(* PLC project TC3_TE1400_GeneratedModule_AdaptiveModel_FB, Beckhoff Automation GmbH & Co. KG TwinCAT 3 Function - TE1400 1.2.1240 *)
(* stored: companyURL www.beckhoff.com, creationDateTime 2022-01-04T00:47:12 *)

TYPE E_TcMatSimDataAreaType : (NotSpecified := 0, Standard, InputSrc, InputDst, OutputSrc, OutputDst, InternalDa, MArea, RetainDa);
END_TYPE

TYPE ST_TcMatSimObjectDataAreaInfo : STRUCT
  pPlcVar : PVOID;
  pModuleProcImg : PVOID;
  nSize : UDINT;
  nDataAreaId : UDINT;
  eDataAreaType : E_TcMatSimDataAreaType;
END_STRUCT;
END_TYPE

{attribute 'pack_mode' := '4'}
TYPE ST_AdaptiveModelInitData : STRUCT
  Header : TComInitDataHdr;
  CallByHdr : TComInitDataElmHdr;
  CallBy : TctModuleCallByType;
  ExecutionSequenceHdr : TComInitDataElmHdr;
  ExecutionSequence : TctModuleExecutionSequenceType;
  StepSizeHdr : TComInitDataElmHdr;
  StepSize : TctStepSizeType;
  ExecuteModelCodeHdr : TComInitDataElmHdr;
  ExecuteModelCode : BOOL;
  ModelParametersHdr : TComInitDataElmHdr;
  ModelParameters : P_AdaptiveModel_T;
  ContextInfoArr_0_TaskOidHdr : TComInitDataElmHdr;
  ContextInfoArr_0_TaskOid : OTCID;
  ContextInfoArr_0_TaskPriorityHdr : TComInitDataElmHdr;
  ContextInfoArr_0_TaskPriority : UDINT;
  ContextInfoArr_0_TaskCycleTimeNsHdr : TComInitDataElmHdr;
  ContextInfoArr_0_TaskCycleTimeNs : UDINT;
  ContextInfoArr_0_TaskPortHdr : TComInitDataElmHdr;
  ContextInfoArr_0_TaskPort : UINT;
  ContextInfoArr_0_TaskSortOrderHdr : TComInitDataElmHdr;
  ContextInfoArr_0_TaskSortOrder : UDINT;
END_STRUCT;
END_TYPE

TYPE ST_AdaptiveModel_Input : STRUCT
  In1 : LREAL;
END_STRUCT;
END_TYPE

TYPE ST_AdaptiveModel_Output : STRUCT
  Out1 : LREAL;
END_STRUCT;
END_TYPE

FUNCTION_BLOCK FB_TcMatSimObject
  VAR_INPUT
    bWriteFbInputValues : BOOL := TRUE;  (* set this flag to write FB input values to the TcComObject's input DataAreas. This will overwrite the mapped input values before module execution. Set to FALSE to read the mapped input values from the TcComObject to the FB. *)
  END_VAR
  VAR
    pDataAreas : POINTER TO ST_TcMatSimObjectDataAreaInfo;  (* process image src and dst pointers and sizes *)
    nDataAreas : UDINT;
    ipObjSrv : ITComObjectServer;  (* global interface pointers *)
    ipTcComObj : ITComObject;  (* object interface pointers *)
    ipTcCyclic : ITcCyclic;
    ipTcPostCyclic : ITcPostCyclic;
    ipTcAdi : ITcADI;
    ipTask : ITcTask;  (* task interface pointers *)
    pInitData : POINTER TO TComInitDataHdr;  (* initial parameters *)
    hResult : HRESULT;  (* hResult of interface calls (0 if no error) *)
    moduleClsId : CLSID;  (* module class ID *)
    assignedClsId : CLSID;  (* expected/desired module class ID *)
    bClassIdVerified : BOOL;
    bDynInstance : BOOL;  (* flag indicating whether the module instance was created dynamically *)
    eInitialObjState : TCOM_STATE := TCOM_STATE.TCOM_STATE_INIT;  (* the object state at the time FB_init was called, FB_exit will try to switch to this state (only if this means to shift down) *)
  END_VAR

            
          

{attribute 'object_name' := 'ReleaseTcComInterface'}
METHOD ReleaseTcComInterface : HRESULT
  VAR
    nStateChangeCnt : DINT := 0;
  END_VAR
                  
IF (ipTcComObj<>0) THEN
  WHILE (State>eInitialObjState AND nStateChangeCnt<1000) DO
    State := eInitialObjState;
    nStateChangeCnt := nStateChangeCnt+1;
  END_WHILE
  ReleaseObjInterfaces();
  IF (bDynInstance) THEN
    ReleaseTcComInterface := TC3_MODULE.FW_ObjMgr_DeleteInstance(ADR(ipTcComObj));
  ELSE
    ipTcComObj.TcRelease();
  END_IF
  ipTcComObj := 0;
END_IF
                  
                
END_METHOD

{attribute 'object_name' := 'ReleaseObjInterfaces'}
METHOD ReleaseObjInterfaces : HRESULT
                  
// release interface pointers
IF (ipTcCyclic<>0) THEN
  ipTcCyclic.TcRelease();
  ipTcCyclic := 0;
END_IF
IF (ipTcPostCyclic<>0) THEN
  ipTcPostCyclic.TcRelease();
  ipTcPostCyclic := 0;
END_IF
IF (ipTcAdi<>0) THEN
  ipTcAdi.TcRelease();
  ipTcAdi := 0;
END_IF
                  
                
END_METHOD

{attribute 'object_name' := 'Internal_SetObjState'}
METHOD Internal_SetObjState
  VAR_INPUT
    hr : REFERENCE TO HRESULT;
    nextState : TCOM_STATE;
  END_VAR
                  
// verify class id
IF (SUCCEEDED(hr)) THEN
  hr := VerifyClassId();
END_IF

// switch object state
IF (SUCCEEDED(hr) AND nextState>=TCOM_STATE_INIT) THEN
  IF (ipTcComObj=0) THEN
    hr := Tc2_System.E_HRESULTAdsErr.NOINTERFACE;
  END_IF
  IF (ipObjSrv=0) THEN
    hr := Tc2_System.E_HRESULTAdsErr.NOINTERFACE;
  END_IF
  IF (SUCCEEDED(hr)) THEN
    hr := ipTcComObj.TcSetObjState(nextState,ipObjSrv,pInitData);
  END_IF
END_IF
                  
                
END_METHOD

{attribute 'object_name' := 'FB_init'}
METHOD FB_init : BOOL
  VAR_INPUT
    bInitRetains : BOOL;  (* init retain variables *)
    bInCopyCode : BOOL;  (* Online Change *)
    oid : OTCID;
  END_VAR
                  
FB_init := SUCCEEDED(Init(oid));
                  
                
END_METHOD

{attribute 'object_name' := 'GetObjPara'}
METHOD GetObjPara : HRESULT
  VAR_INPUT
    pid : PTCID;
    nData : UDINT;
    pData : PVOID;
  END_VAR
                  
IF (ipTcComObj=0) THEN
  GetObjPara := Tc2_System.E_HRESULTAdsErr.NOINTERFACE;
END_IF

IF (SUCCEEDED(GetObjPara)) THEN
  GetObjPara := ipTcComObj.TcGetObjPara(pid:=pid,nData,pData,0);
END_IF
                  
                
END_METHOD

{attribute 'object_name' := 'QueryObjInterface'}
METHOD QueryObjInterface
  VAR_INPUT
    hr : REFERENCE TO HRESULT;
    iid : REFERENCE TO IID;
    pipItf : POINTER TO ITcUnknown;
  END_VAR
  VAR CONSTANT
    pNull : PVOID := 0;
  END_VAR
                  
IF (SUCCEEDED(hr)) THEN
  IF (ipTcComObj=0) THEN
    hr := Tc2_System.E_HRESULTAdsErr.NOINTERFACE;
  ELSIF (pipItf^=ULINT_TO_DWORD(pNull)) THEN
    hr := ipTcComObj.TcQueryInterface(iid:= iid, pipItf:=pipItf);
  END_IF
END_IF
                  
                
END_METHOD

{attribute 'object_name' := 'SaveOnlineParametersForInit'}
METHOD SaveOnlineParametersForInit : HRESULT
  VAR
    idx : UINT;
    pInitElemHdr : POINTER TO TComInitDataElmHdr;
    pData : PVOID;
    nData : UDINT;
  END_VAR
  VAR CONSTANT
    nInitDataAlignment : UDINT := 4;
  END_VAR
                  IF (pInitData<>0) THEN
  pInitElemHdr := pInitData + SIZEOF(pInitData^);
  FOR idx:=1 TO pInitData^.uiElmCnt DO
    pData := pInitElemHdr + ULINT_TO_DWORD(SIZEOF(pInitElemHdr^));
    nData := pInitElemHdr^.cbData;
    SaveOnlineParametersForInit := GetObjPara(pInitElemHdr^.indexOffset,nData,pData);
    IF (FAILED(SaveOnlineParametersForInit)) THEN
      RETURN;
    END_IF
    pInitElemHdr := pData + (nInitDataAlignment*((nData + nInitDataAlignment - 1)/nInitDataAlignment));
  END_FOR
ELSE
	SaveOnlineParametersForInit := Tc2_System.E_HRESULTAdsErr.NOTINIT;
END_IF
                  
                
END_METHOD

{attribute 'object_name' := 'ResetHresult'}
METHOD ResetHresult
                  hResult := S_OK;
                
END_METHOD

{attribute 'object_name' := 'Execute'}
METHOD Execute : HRESULT
  VAR
    nDaIdx : UDINT;
    pCurDataArea : POINTER TO ST_TcMatSimObjectDataAreaInfo;
  END_VAR
                  
IF (SUCCEEDED(hResult)) THEN
  hResult := VerifyClassId();
END_IF

IF (SUCCEEDED(hResult) AND State<>TCOM_STATE_OP) THEN
  hResult := Tc2_System.E_HRESULTAdsErr.NOTREADY;
END_IF

// get image pointers
IF (SUCCEEDED(hResult)) THEN
  GetImagePtrs(hResult);
END_IF

// copy inputs
IF (pDataAreas<>0 AND nDataAreas>0 AND bWriteFbInputValues) THEN
  FOR nDaIdx:=0 TO nDataAreas-1 DO
    IF (FAILED(hResult))THEN
      CONTINUE;
    END_IF
    pCurDataArea := pDataAreas + nDaIdx*SIZEOF(ST_TcMatSimObjectDataAreaInfo);
    IF ((pCurDataArea^.eDataAreaType <> E_TcMatSimDataAreaType.InputDst))THEN
      CONTINUE;
    END_IF
    IF (pCurDataArea^.pModuleProcImg<>0 AND pCurDataArea^.pPlcVar<>0) THEN
      MEMCPY(pCurDataArea^.pModuleProcImg,pCurDataArea^.pPlcVar,pCurDataArea^.nSize);
    ELSE
      hResult := Tc2_System.E_HRESULTAdsErr.NOINTERFACE;
    END_IF
  END_FOR
END_IF

// call cycle update
IF (SUCCEEDED(hResult)) THEN
  IF (ipTcCyclic<>0) THEN
    hResult := ipTcCyclic.CycleUpdate(ipTask:= ipTask, ipCaller:= 0, context:= 0);
  ELSE
    hResult := Tc2_System.E_HRESULTAdsErr.NOINTERFACE;
  END_IF
END_IF

// copy outputs
IF (pDataAreas<>0 AND nDataAreas>0) THEN
  FOR nDaIdx:=0 TO nDataAreas-1 DO
    IF (FAILED(hResult))THEN
      CONTINUE;
    END_IF
    pCurDataArea := pDataAreas + nDaIdx*SIZEOF(ST_TcMatSimObjectDataAreaInfo);
    IF ((pCurDataArea^.eDataAreaType = E_TcMatSimDataAreaType.OutputSrc) OR NOT bWriteFbInputValues) THEN
      IF (pCurDataArea^.pModuleProcImg<>0 AND pCurDataArea^.pPlcVar<>0) THEN
        MEMCPY(pCurDataArea^.pPlcVar,pCurDataArea^.pModuleProcImg,pCurDataArea^.nSize);
      ELSE
        hResult := Tc2_System.E_HRESULTAdsErr.NOINTERFACE;
      END_IF
    END_IF
  END_FOR
END_IF


// call post cyclic update
IF (SUCCEEDED(hResult)) THEN
  IF (ipTcPostCyclic<>0) THEN
    hResult := ipTcPostCyclic.PostCyclicUpdate(ipTask:= 0, ipCaller:= 0, context:= 0);
  ELSE
    hResult := Tc2_System.E_HRESULTAdsErr.NOINTERFACE;
  END_IF
END_IF

ReleaseImagePtrs();

Execute := hResult;
                  
                
END_METHOD

{attribute 'object_name' := 'GetImagePtrs'}
METHOD GetImagePtrs
  VAR_INPUT
    hr : REFERENCE TO HRESULT;
  END_VAR
  VAR
    nDaIdx : UDINT;
    pCurDataArea : POINTER TO ST_TcMatSimObjectDataAreaInfo;
  END_VAR
                  
IF (ipTcAdi=0) THEN
  hr := Tc2_System.E_HRESULTAdsErr.NOINTERFACE;
END_IF
IF(State<>TCOM_STATE_OP)THEN
  hr := Tc2_System.E_HRESULTAdsErr.INVALIDSTATE;
END_IF


// get pointers to process images
IF (pDataAreas<>0 AND nDataAreas>0) THEN
  FOR nDaIdx:=0 TO nDataAreas-1 DO
    pCurDataArea := pDataAreas + nDaIdx*SIZEOF(ST_TcMatSimObjectDataAreaInfo);
    IF (FAILED(hr))THEN
      CONTINUE;
    END_IF
    IF ((pCurDataArea^.eDataAreaType <> E_TcMatSimDataAreaType.InputDst) AND (pCurDataArea^.eDataAreaType <> E_TcMatSimDataAreaType.OutputSrc))THEN
      CONTINUE;
    END_IF
    IF (pCurDataArea^.pModuleProcImg=0 AND pCurDataArea^.nSize>0) THEN
      hr := ipTcAdi.GetImagePtr(size:= pCurDataArea^.nSize , offs:=0 , adi_x:=pCurDataArea^.nDataAreaId , ppData:=ADR(pCurDataArea^.pModuleProcImg));
    END_IF
  END_FOR
END_IF

IF (FAILED(hr)) THEN
  ReleaseImagePtrs();
END_IF
                  
                
END_METHOD

{attribute 'object_name' := 'VerifyClassId'}
METHOD VerifyClassId : HRESULT
  VAR
    emptyClsId : CLSID;
  END_VAR
                  memset(ADR(emptyClsId),0,SIZEOF(emptyClsId));
IF (bClassIdVerified) THEN
  // class ID was already verified
  VerifyClassId := Tc2_System.E_HRESULTAdsErr.HRESULT_ADS_NOERROR;
ELSIF (memcmp(ADR(assignedClsId),ADR(emptyClsId),SIZEOF(assignedClsId))=0) THEN
  // skip class ID verification if no assignedClsId specified
  VerifyClassId := Tc2_System.E_HRESULTAdsErr.HRESULT_ADS_NOERROR;
ELSE
  // verify class ID
  VerifyClassId := ReadModuleClassId();

  IF (SUCCEEDED(VerifyClassId)) THEN
    IF (memcmp(ADR(assignedClsId),ADR(moduleClsId),SIZEOF(assignedClsId))<>0) THEN
     VerifyClassId := Tc2_System.E_HRESULTAdsErr.INVALIDCLSID;
    END_IF
  END_IF
  bClassIdVerified := SUCCEEDED(VerifyClassId);
END_IF
                  
                
END_METHOD

{attribute 'object_name' := 'SetObjPara'}
METHOD SetObjPara : HRESULT
  VAR_INPUT
    pid : PTCID;
    nData : UDINT;
    pData : PVOID;
  END_VAR
                  
IF (ipTcComObj=0) THEN
  SetObjPara := Tc2_System.E_HRESULTAdsErr.NOINTERFACE;
END_IF

IF (SUCCEEDED(SetObjPara)) THEN
  SetObjPara := ipTcComObj.TcSetObjPara(pid:=pid,nData,pData,0);
END_IF
                  
                
END_METHOD

{attribute 'object_name' := 'QueryTcComInterface'}
METHOD QueryTcComInterface
  VAR_INPUT
    hr : REFERENCE TO HRESULT;
    oid : OTCID;
  END_VAR
                  
IF (ipObjSrv=0) THEN
  hr := Tc2_System.E_HRESULTAdsErr.NOINTERFACE;
END_IF

IF (SUCCEEDED(hr) AND ipTcComObj=0) THEN
  bDynInstance := FALSE;
  IF(oid>0) THEN
    // query interface of existing object
    hr := ipObjSrv.TcQueryObjectInterface(oid,IID_ITComObject,ADR(ipTcComObj));
  ELSE
    // create new instance and get the object interface
    hr := ipObjSrv.TcCreateInstance(assignedClsId,IID_ITComObject,ADR(ipTcComObj));
    IF (SUCCEEDED(hr)) THEN
      bDynInstance := TRUE;
      hr := ipTcComObj.TcSetObjectId(OTCID_CreateNewId);
    END_IF
  END_IF
  IF (SUCCEEDED(hr)) THEN
    eInitialObjState := State;
  END_IF
END_IF
                  
                
END_METHOD

{attribute 'object_name' := 'ReleaseImagePtrs'}
METHOD ReleaseImagePtrs : HRESULT
  VAR
    nDaIdx : UDINT;
    pCurDataArea : POINTER TO ST_TcMatSimObjectDataAreaInfo;
  END_VAR
                  
IF (ipTcAdi=0) THEN
  ReleaseImagePtrs := Tc2_System.E_HRESULTAdsErr.NOINTERFACE;
END_IF

IF (SUCCEEDED(ReleaseImagePtrs) AND pDataAreas<>0 AND nDataAreas>0) THEN
  // release pointers to the simulink module process images
  FOR nDaIdx:=0 TO nDataAreas-1 DO
    pCurDataArea := pDataAreas + nDaIdx*SIZEOF(ST_TcMatSimObjectDataAreaInfo);

    IF (pCurDataArea^.pModuleProcImg<>0) THEN
      ipTcAdi.ReleaseImagePtr(pData:=pCurDataArea^.pModuleProcImg);
      pCurDataArea^.pModuleProcImg := 0;
    END_IF
  END_FOR
END_IF
                  
                
END_METHOD

{attribute 'object_name' := 'FB_exit'}
METHOD FB_exit : BOOL
  VAR_INPUT
    bInCopyCode : BOOL;  (* Online Change *)
  END_VAR
                  
IF (NOT bInCopyCode) THEN
  IF (ipObjSrv<>0) THEN
    ipObjSrv.TcRelease();
    ipObjSrv := 0;
  END_IF

  ReleaseTcComInterface();
END_IF
                  
                
END_METHOD

{attribute 'object_name' := 'InitObjName'}
METHOD InitObjName
  VAR_INPUT
    hr : REFERENCE TO HRESULT;
  END_VAR
  VAR
    objectName : STRING(255) := 'TcMatSimObject_PlcRtFbInstance';
    oid : OTCID;
  END_VAR
                  
IF (SUCCEEDED(hr)) THEN
  hr := ipTcComObj.TcGetObjectId(oid);
END_IF

IF (SUCCEEDED(hr) and bDynInstance) THEN
  objectName := TC2_STANDARD.CONCAT(objectName,'_');
  objectName := TC2_STANDARD.CONCAT(objectName,UDINT_TO_STRING(oid));
  hr := ipTcComObj.TcSetObjectName(ADR(objectName));
END_IF
                  
                
END_METHOD

{attribute 'object_name' := 'SetObjState'}
METHOD SetObjState : HRESULT
  VAR_INPUT
    finalState : TCOM_STATE;
  END_VAR
  VAR
    bShiftUp : BOOL;
    bShiftDown : BOOL;
    currentState : TCOM_STATE;
  END_VAR
                  
currentState := State;

bShiftUp := finalState>currentState;
bShiftDown := finalState<currentState;

// do not switch up on error
IF (FAILED(hresult)) THEN
  bShiftUp := FALSE;
END_IF
// reset existing error on switching down
IF (bShiftDown) THEN
  ResetHresult();
END_IF

// prepared state switch
CASE currentState OF
  TCOM_STATE_INIT:
    IF(bShiftUp) THEN
      QueryTcComInterface(hResult,0);
      Internal_SetObjState(hResult,TCOM_STATE.TCOM_STATE_PREOP);
      InitObjName(hResult);
    END_IF

  TCOM_STATE_PREOP:
    IF(bShiftUp) THEN
      Internal_SetObjState(hResult,TCOM_STATE.TCOM_STATE_SAFEOP);
      QueryObjInterfaces(hResult);
    ELSIF (bShiftDown) THEN
      Internal_SetObjState(hResult,TCOM_STATE.TCOM_STATE_INIT);
    END_IF

  TCOM_STATE_SAFEOP:
    IF(bShiftUp) THEN
      Internal_SetObjState(hResult,TCOM_STATE.TCOM_STATE_OP);
      QueryObjInterfaces(hResult);
    ELSIF (bShiftDown) THEN
      Internal_SetObjState(hResult,TCOM_STATE.TCOM_STATE_PREOP);
      ReleaseObjInterfaces();
    END_IF


  TCOM_STATE_OP:
    IF (bShiftDown) THEN
      Internal_SetObjState(hResult,TCOM_STATE.TCOM_STATE_SAFEOP);
    END_IF
END_CASE

SetObjState := hResult;
                  
                
END_METHOD

{attribute 'object_name' := 'QueryObjInterfaces'}
METHOD QueryObjInterfaces
  VAR_INPUT
    hr : REFERENCE TO HRESULT;
  END_VAR
                  
IF(State<TCOM_STATE_PREOP)THEN
  hr := Tc2_System.E_HRESULTAdsErr.INVALIDSTATE;
END_IF

//cyclic interface
QueryObjInterface(hr,IID_ITCCYCLIC,ADR(ipTcCyclic));
//post cyclic interface
QueryObjInterface(hr,IID_ITCPOSTCYCLIC,ADR(ipTcPostCyclic));
//adi interface
QueryObjInterface(hr,IID_ITcADI,ADR(ipTcAdi));
                  
                
END_METHOD

{attribute 'object_name' := 'Init'}
METHOD Init : HRESULT
  VAR_INPUT
    oid : OTCID;
  END_VAR
                  
// preinitialize variables
memset(ADR(moduleClsId),0,SIZEOF(moduleClsId));
bClassIdVerified := FALSE;
hResult := Tc2_System.E_HRESULTAdsErr.HRESULT_ADS_NOERROR;

// get object server
IF (ipObjSrv=0) THEN
  hResult := FW_ObjMgr_GetObjectServer(_AppInfo.ObjId,ADR(ipObjSrv));
END_IF

// try to get object interfaces
IF (SUCCEEDED(hresult)) THEN
  QueryTcComInterface(hResult,oid);
END_IF

// verify class id
IF (SUCCEEDED(hresult)) THEN
  hresult := VerifyClassId();
END_IF

// query interfaces, if the current state is higher than INIT
IF (SUCCEEDED(hresult) AND State>TCOM_STATE.TCOM_STATE_INIT) THEN
  QueryObjInterfaces(hResult);
END_IF

// return value
Init := hresult;
                  
                
END_METHOD

{attribute 'object_name' := 'ReadModuleClassId'}
METHOD ReadModuleClassId : HRESULT
  VAR
    emptyClsId : CLSID;
  END_VAR
                  memset(ADR(emptyClsId),0,SIZEOF(emptyClsId));
IF (memcmp(ADR(moduleClsId),ADR(emptyClsId),SIZEOF(moduleClsId))=0) THEN
  IF (ipTcComObj=0) THEN
    ReadModuleClassId := Tc2_System.E_HRESULTAdsErr.NOINTERFACE;
  END_IF

  //objectClsId := clsid;
  IF (SUCCEEDED(ReadModuleClassId)) THEN
    ReadModuleClassId := ipTcComObj.GetClassId(moduleClsId);
  END_IF
END_IF
                
END_METHOD

METHOD PUBLIC AssignClassId
VAR_INPUT
	clsId : CLSID;
END_VAR
                  assignedClsId := clsId;
bClassIdVerified := false;
                  
                
END_METHOD

PROPERTY Error : BOOL
GET
                    Error := FAILED(hResult);
                  
END_GET
END_PROPERTY

METHOD PUBLIC SetDataAreaInfo
VAR_INPUT
  pDataAreas: POINTER TO ST_TcMatSimObjectDataAreaInfo;
  nDataAreas: UDINT;
END_VAR
                  
THIS^.nDataAreas := nDataAreas;
THIS^.pDataAreas := pDataAreas;
                  
                
END_METHOD

METHOD PUBLIC SetInitDataInfo
VAR_INPUT
  pInitData : POINTER TO TComInitDataHdr;
END_VAR
                  this^.pInitData := pInitData;
                
END_METHOD

PROPERTY ClassId : CLSID
GET
                    hResult := ReadModuleClassId();
ClassId := moduleClsId;
                    
                  
END_GET
END_PROPERTY

PROPERTY State : TCOM_STATE
GET
  VAR
    hr : HRESULT := S_OK;
    eObjState : TCOM_STATE;
  END_VAR
                    
IF (ipTcComObj<>0) THEN
  hr := ipTcComObj.TcGetObjState(ADR(eObjState));
IF (FAILED(hr)) THEN
  eObjState := TCOM_STATE.TCOM_STATE_INIT;
END_IF
ELSE
  eObjState := TCOM_STATE.TCOM_STATE_INIT;
END_IF
State := eObjState;
                    
                  
END_GET
SET
                    SetObjState(State);
                  
END_SET
END_PROPERTY

PROPERTY ErrorCode : HRESULT
GET
                    ErrorCode := hResult;
                  
END_GET
END_PROPERTY
END_FUNCTION_BLOCK

{attribute 'TcDependOnClassFactory' := 'AdaptiveModel'}
FUNCTION_BLOCK FB_AdaptiveModel EXTENDS FB_TcMatSimObject
  VAR_INPUT
    stInput : ST_AdaptiveModel_Input;
  END_VAR
  VAR_OUTPUT
    stOutput : ST_AdaptiveModel_Output;
  END_VAR
  VAR
    stInitData : ST_AdaptiveModelInitData;
    arrDataAreas : ARRAY[1..2] OF ST_TcMatSimObjectDataAreaInfo;
    bParametersVerified : BOOL;
  END_VAR

            
          

{attribute 'object_name' := 'Internal_SetObjState'}
METHOD Internal_SetObjState
  VAR_INPUT
    hr : REFERENCE TO HRESULT;
    nextState : TCOM_STATE;
  END_VAR
                  
// update pointer to InitData structure
SetInitDataInfo(ADR(stInitData));
// call base method
SUPER^.Internal_SetObjState(hr,nextState);
                  
                
END_METHOD

{attribute 'object_name' := 'SaveOnlineParametersForInit'}
METHOD SaveOnlineParametersForInit : HRESULT
  VAR
    idx : UINT;
    pInitElemHdr : POINTER TO TComInitDataElmHdr;
    pData : PVOID;
    nData : UDINT;
  END_VAR
  VAR CONSTANT
    nInitDataAlignment : UDINT := 4;
  END_VAR
                  
// update pointer to InitData structure
SetInitDataInfo(ADR(stInitData));
// call base method
SaveOnlineParametersForInit := SUPER^.SaveOnlineParametersForInit();
                  
                
END_METHOD

METHOD FB_init : BOOL
  VAR_INPUT
    bInitRetains : BOOL;  (* if TRUE, the retain variables are initialized (warm start / cold start) *)
    bInCopyCode : BOOL;  (* if TRUE, the instance afterwards gets moved into the copy code (online change) *)
    oid : OTCID;
  END_VAR
  VAR
    clsId : CLSID;
  END_VAR
                  
// initialize flags
bParametersVerified := false;
                    
// set module class id for compatibility check
clsId.Data1 := 16#dc3905a3;
clsId.Data2 := 16#3c10;
clsId.Data3 := 16#463f;
clsId.Data4[0] := 16#97;
clsId.Data4[1] := 16#74;
clsId.Data4[2] := 16#0a;
clsId.Data4[3] := 16#63;
clsId.Data4[4] := 16#82;
clsId.Data4[5] := 16#3c;
clsId.Data4[6] := 16#f9;
clsId.Data4[7] := 16#4a;

AssignClassId(clsId);
                    
// initialize InitData structure with default values              
stInitData.CallByHdr.indexGroup := 0;
stInitData.CallByHdr.indexOffset := 16#00000000;
stInitData.CallByHdr.cbData := SIZEOF(stInitData.CallBy);
stInitData.CallBy := TctModuleCallByType.Module;
stInitData.ExecutionSequenceHdr.indexGroup := 0;
stInitData.ExecutionSequenceHdr.indexOffset := 16#00000001;
stInitData.ExecutionSequenceHdr.cbData := SIZEOF(stInitData.ExecutionSequence);
stInitData.ExecutionSequence := TctModuleExecutionSequenceType.StateUpdateAfterOutputMapping;
stInitData.StepSizeHdr.indexGroup := 0;
stInitData.StepSizeHdr.indexOffset := 16#00000002;
stInitData.StepSizeHdr.cbData := SIZEOF(stInitData.StepSize);
stInitData.StepSize := TctStepSizeType.RequireMatchingTaskCycleTime;
stInitData.ExecuteModelCodeHdr.indexGroup := 0;
stInitData.ExecuteModelCodeHdr.indexOffset := 16#00000007;
stInitData.ExecuteModelCodeHdr.cbData := SIZEOF(stInitData.ExecuteModelCode);
stInitData.ExecuteModelCode := 1;
stInitData.ModelParametersHdr.indexGroup := 0;
stInitData.ModelParametersHdr.indexOffset := 16#83000000;
stInitData.ModelParametersHdr.cbData := SIZEOF(stInitData.ModelParameters);
stInitData.ModelParameters.A_01 := 20;
stInitData.ModelParameters.a := 2;
stInitData.ModelParameters.b := 5;
stInitData.ModelParameters.DefuzzifyOutputs_SimulateUsing := 1;
stInitData.ModelParameters.EvaluateRuleAntecedents_Simulat := 1;
stInitData.ModelParameters.EvaluateRuleConsequents_Simulat := 1;
stInitData.ModelParameters.OutputSamplePoints_Value[0] := -6;
stInitData.ModelParameters.OutputSamplePoints_Value[1] := -6;
stInitData.ModelParameters.OutputSamplePoints_Value[2] := -6;
stInitData.ModelParameters.OutputSamplePoints_Value[3] := -5.8799999999999999;
stInitData.ModelParameters.OutputSamplePoints_Value[4] := -5.8799999999999999;
stInitData.ModelParameters.OutputSamplePoints_Value[5] := -5.8799999999999999;
stInitData.ModelParameters.OutputSamplePoints_Value[6] := -5.7599999999999998;
stInitData.ModelParameters.OutputSamplePoints_Value[7] := -5.7599999999999998;
stInitData.ModelParameters.OutputSamplePoints_Value[8] := -5.7599999999999998;
stInitData.ModelParameters.OutputSamplePoints_Value[9] := -5.6399999999999997;
stInitData.ModelParameters.OutputSamplePoints_Value[10] := -5.6399999999999997;
stInitData.ModelParameters.OutputSamplePoints_Value[11] := -5.6399999999999997;
stInitData.ModelParameters.OutputSamplePoints_Value[12] := -5.5199999999999996;
stInitData.ModelParameters.OutputSamplePoints_Value[13] := -5.5199999999999996;
stInitData.ModelParameters.OutputSamplePoints_Value[14] := -5.5199999999999996;
stInitData.ModelParameters.OutputSamplePoints_Value[15] := -5.4000000000000004;
stInitData.ModelParameters.OutputSamplePoints_Value[16] := -5.4000000000000004;
stInitData.ModelParameters.OutputSamplePoints_Value[17] := -5.4000000000000004;
stInitData.ModelParameters.OutputSamplePoints_Value[18] := -5.2800000000000002;
stInitData.ModelParameters.OutputSamplePoints_Value[19] := -5.2800000000000002;
stInitData.ModelParameters.OutputSamplePoints_Value[20] := -5.2800000000000002;
stInitData.ModelParameters.OutputSamplePoints_Value[21] := -5.1600000000000001;
stInitData.ModelParameters.OutputSamplePoints_Value[22] := -5.1600000000000001;
stInitData.ModelParameters.OutputSamplePoints_Value[23] := -5.1600000000000001;
stInitData.ModelParameters.OutputSamplePoints_Value[24] := -5.04;
stInitData.ModelParameters.OutputSamplePoints_Value[25] := -5.04;
stInitData.ModelParameters.OutputSamplePoints_Value[26] := -5.04;
stInitData.ModelParameters.OutputSamplePoints_Value[27] := -4.9199999999999999;
stInitData.ModelParameters.OutputSamplePoints_Value[28] := -4.9199999999999999;
stInitData.ModelParameters.OutputSamplePoints_Value[29] := -4.9199999999999999;
stInitData.ModelParameters.OutputSamplePoints_Value[30] := -4.7999999999999998;
stInitData.ModelParameters.OutputSamplePoints_Value[31] := -4.7999999999999998;
stInitData.ModelParameters.OutputSamplePoints_Value[32] := -4.7999999999999998;
stInitData.ModelParameters.OutputSamplePoints_Value[33] := -4.6799999999999997;
stInitData.ModelParameters.OutputSamplePoints_Value[34] := -4.6799999999999997;
stInitData.ModelParameters.OutputSamplePoints_Value[35] := -4.6799999999999997;
stInitData.ModelParameters.OutputSamplePoints_Value[36] := -4.5600000000000005;
stInitData.ModelParameters.OutputSamplePoints_Value[37] := -4.5600000000000005;
stInitData.ModelParameters.OutputSamplePoints_Value[38] := -4.5600000000000005;
stInitData.ModelParameters.OutputSamplePoints_Value[39] := -4.4399999999999995;
stInitData.ModelParameters.OutputSamplePoints_Value[40] := -4.4399999999999995;
stInitData.ModelParameters.OutputSamplePoints_Value[41] := -4.4399999999999995;
stInitData.ModelParameters.OutputSamplePoints_Value[42] := -4.3200000000000003;
stInitData.ModelParameters.OutputSamplePoints_Value[43] := -4.3200000000000003;
stInitData.ModelParameters.OutputSamplePoints_Value[44] := -4.3200000000000003;
stInitData.ModelParameters.OutputSamplePoints_Value[45] := -4.2000000000000002;
stInitData.ModelParameters.OutputSamplePoints_Value[46] := -4.2000000000000002;
stInitData.ModelParameters.OutputSamplePoints_Value[47] := -4.2000000000000002;
stInitData.ModelParameters.OutputSamplePoints_Value[48] := -4.0800000000000001;
stInitData.ModelParameters.OutputSamplePoints_Value[49] := -4.0800000000000001;
stInitData.ModelParameters.OutputSamplePoints_Value[50] := -4.0800000000000001;
stInitData.ModelParameters.OutputSamplePoints_Value[51] := -3.96;
stInitData.ModelParameters.OutputSamplePoints_Value[52] := -3.96;
stInitData.ModelParameters.OutputSamplePoints_Value[53] := -3.96;
stInitData.ModelParameters.OutputSamplePoints_Value[54] := -3.8399999999999999;
stInitData.ModelParameters.OutputSamplePoints_Value[55] := -3.8399999999999999;
stInitData.ModelParameters.OutputSamplePoints_Value[56] := -3.8399999999999999;
stInitData.ModelParameters.OutputSamplePoints_Value[57] := -3.7200000000000002;
stInitData.ModelParameters.OutputSamplePoints_Value[58] := -3.7200000000000002;
stInitData.ModelParameters.OutputSamplePoints_Value[59] := -3.7200000000000002;
stInitData.ModelParameters.OutputSamplePoints_Value[60] := -3.6000000000000001;
stInitData.ModelParameters.OutputSamplePoints_Value[61] := -3.6000000000000001;
stInitData.ModelParameters.OutputSamplePoints_Value[62] := -3.6000000000000001;
stInitData.ModelParameters.OutputSamplePoints_Value[63] := -3.48;
stInitData.ModelParameters.OutputSamplePoints_Value[64] := -3.48;
stInitData.ModelParameters.OutputSamplePoints_Value[65] := -3.48;
stInitData.ModelParameters.OutputSamplePoints_Value[66] := -3.3599999999999999;
stInitData.ModelParameters.OutputSamplePoints_Value[67] := -3.3599999999999999;
stInitData.ModelParameters.OutputSamplePoints_Value[68] := -3.3599999999999999;
stInitData.ModelParameters.OutputSamplePoints_Value[69] := -3.2400000000000002;
stInitData.ModelParameters.OutputSamplePoints_Value[70] := -3.2400000000000002;
stInitData.ModelParameters.OutputSamplePoints_Value[71] := -3.2400000000000002;
stInitData.ModelParameters.OutputSamplePoints_Value[72] := -3.1200000000000001;
stInitData.ModelParameters.OutputSamplePoints_Value[73] := -3.1200000000000001;
stInitData.ModelParameters.OutputSamplePoints_Value[74] := -3.1200000000000001;
stInitData.ModelParameters.OutputSamplePoints_Value[75] := -3;
stInitData.ModelParameters.OutputSamplePoints_Value[76] := -3;
stInitData.ModelParameters.OutputSamplePoints_Value[77] := -3;
stInitData.ModelParameters.OutputSamplePoints_Value[78] := -2.8799999999999999;
stInitData.ModelParameters.OutputSamplePoints_Value[79] := -2.8799999999999999;
stInitData.ModelParameters.OutputSamplePoints_Value[80] := -2.8799999999999999;
stInitData.ModelParameters.OutputSamplePoints_Value[81] := -2.7599999999999998;
stInitData.ModelParameters.OutputSamplePoints_Value[82] := -2.7599999999999998;
stInitData.ModelParameters.OutputSamplePoints_Value[83] := -2.7599999999999998;
stInitData.ModelParameters.OutputSamplePoints_Value[84] := -2.6400000000000001;
stInitData.ModelParameters.OutputSamplePoints_Value[85] := -2.6400000000000001;
stInitData.ModelParameters.OutputSamplePoints_Value[86] := -2.6400000000000001;
stInitData.ModelParameters.OutputSamplePoints_Value[87] := -2.52;
stInitData.ModelParameters.OutputSamplePoints_Value[88] := -2.52;
stInitData.ModelParameters.OutputSamplePoints_Value[89] := -2.52;
stInitData.ModelParameters.OutputSamplePoints_Value[90] := -2.3999999999999999;
stInitData.ModelParameters.OutputSamplePoints_Value[91] := -2.3999999999999999;
stInitData.ModelParameters.OutputSamplePoints_Value[92] := -2.3999999999999999;
stInitData.ModelParameters.OutputSamplePoints_Value[93] := -2.2799999999999998;
stInitData.ModelParameters.OutputSamplePoints_Value[94] := -2.2799999999999998;
stInitData.ModelParameters.OutputSamplePoints_Value[95] := -2.2799999999999998;
stInitData.ModelParameters.OutputSamplePoints_Value[96] := -2.1600000000000001;
stInitData.ModelParameters.OutputSamplePoints_Value[97] := -2.1600000000000001;
stInitData.ModelParameters.OutputSamplePoints_Value[98] := -2.1600000000000001;
stInitData.ModelParameters.OutputSamplePoints_Value[99] := -2.04;
stInitData.ModelParameters.OutputSamplePoints_Value[100] := -2.04;
stInitData.ModelParameters.OutputSamplePoints_Value[101] := -2.04;
stInitData.ModelParameters.OutputSamplePoints_Value[102] := -1.9199999999999999;
stInitData.ModelParameters.OutputSamplePoints_Value[103] := -1.9199999999999999;
stInitData.ModelParameters.OutputSamplePoints_Value[104] := -1.9199999999999999;
stInitData.ModelParameters.OutputSamplePoints_Value[105] := -1.7999999999999998;
stInitData.ModelParameters.OutputSamplePoints_Value[106] := -1.7999999999999998;
stInitData.ModelParameters.OutputSamplePoints_Value[107] := -1.7999999999999998;
stInitData.ModelParameters.OutputSamplePoints_Value[108] := -1.6799999999999997;
stInitData.ModelParameters.OutputSamplePoints_Value[109] := -1.6799999999999997;
stInitData.ModelParameters.OutputSamplePoints_Value[110] := -1.6799999999999997;
stInitData.ModelParameters.OutputSamplePoints_Value[111] := -1.5599999999999996;
stInitData.ModelParameters.OutputSamplePoints_Value[112] := -1.5599999999999996;
stInitData.ModelParameters.OutputSamplePoints_Value[113] := -1.5599999999999996;
stInitData.ModelParameters.OutputSamplePoints_Value[114] := -1.4400000000000004;
stInitData.ModelParameters.OutputSamplePoints_Value[115] := -1.4400000000000004;
stInitData.ModelParameters.OutputSamplePoints_Value[116] := -1.4400000000000004;
stInitData.ModelParameters.OutputSamplePoints_Value[117] := -1.3200000000000003;
stInitData.ModelParameters.OutputSamplePoints_Value[118] := -1.3200000000000003;
stInitData.ModelParameters.OutputSamplePoints_Value[119] := -1.3200000000000003;
stInitData.ModelParameters.OutputSamplePoints_Value[120] := -1.2000000000000002;
stInitData.ModelParameters.OutputSamplePoints_Value[121] := -1.2000000000000002;
stInitData.ModelParameters.OutputSamplePoints_Value[122] := -1.2000000000000002;
stInitData.ModelParameters.OutputSamplePoints_Value[123] := -1.0800000000000001;
stInitData.ModelParameters.OutputSamplePoints_Value[124] := -1.0800000000000001;
stInitData.ModelParameters.OutputSamplePoints_Value[125] := -1.0800000000000001;
stInitData.ModelParameters.OutputSamplePoints_Value[126] := -0.95999999999999996;
stInitData.ModelParameters.OutputSamplePoints_Value[127] := -0.95999999999999996;
stInitData.ModelParameters.OutputSamplePoints_Value[128] := -0.95999999999999996;
stInitData.ModelParameters.OutputSamplePoints_Value[129] := -0.83999999999999986;
stInitData.ModelParameters.OutputSamplePoints_Value[130] := -0.83999999999999986;
stInitData.ModelParameters.OutputSamplePoints_Value[131] := -0.83999999999999986;
stInitData.ModelParameters.OutputSamplePoints_Value[132] := -0.71999999999999975;
stInitData.ModelParameters.OutputSamplePoints_Value[133] := -0.71999999999999975;
stInitData.ModelParameters.OutputSamplePoints_Value[134] := -0.71999999999999975;
stInitData.ModelParameters.OutputSamplePoints_Value[135] := -0.59999999999999964;
stInitData.ModelParameters.OutputSamplePoints_Value[136] := -0.59999999999999964;
stInitData.ModelParameters.OutputSamplePoints_Value[137] := -0.59999999999999964;
stInitData.ModelParameters.OutputSamplePoints_Value[138] := -0.48000000000000043;
stInitData.ModelParameters.OutputSamplePoints_Value[139] := -0.48000000000000043;
stInitData.ModelParameters.OutputSamplePoints_Value[140] := -0.48000000000000043;
stInitData.ModelParameters.OutputSamplePoints_Value[141] := -0.36000000000000032;
stInitData.ModelParameters.OutputSamplePoints_Value[142] := -0.36000000000000032;
stInitData.ModelParameters.OutputSamplePoints_Value[143] := -0.36000000000000032;
stInitData.ModelParameters.OutputSamplePoints_Value[144] := -0.24000000000000021;
stInitData.ModelParameters.OutputSamplePoints_Value[145] := -0.24000000000000021;
stInitData.ModelParameters.OutputSamplePoints_Value[146] := -0.24000000000000021;
stInitData.ModelParameters.OutputSamplePoints_Value[147] := -0.12000000000000011;
stInitData.ModelParameters.OutputSamplePoints_Value[148] := -0.12000000000000011;
stInitData.ModelParameters.OutputSamplePoints_Value[149] := -0.12000000000000011;
stInitData.ModelParameters.OutputSamplePoints_Value[150] := 0;
stInitData.ModelParameters.OutputSamplePoints_Value[151] := 0;
stInitData.ModelParameters.OutputSamplePoints_Value[152] := 0;
stInitData.ModelParameters.OutputSamplePoints_Value[153] := 0.12000000000000011;
stInitData.ModelParameters.OutputSamplePoints_Value[154] := 0.12000000000000011;
stInitData.ModelParameters.OutputSamplePoints_Value[155] := 0.12000000000000011;
stInitData.ModelParameters.OutputSamplePoints_Value[156] := 0.24000000000000021;
stInitData.ModelParameters.OutputSamplePoints_Value[157] := 0.24000000000000021;
stInitData.ModelParameters.OutputSamplePoints_Value[158] := 0.24000000000000021;
stInitData.ModelParameters.OutputSamplePoints_Value[159] := 0.36000000000000032;
stInitData.ModelParameters.OutputSamplePoints_Value[160] := 0.36000000000000032;
stInitData.ModelParameters.OutputSamplePoints_Value[161] := 0.36000000000000032;
stInitData.ModelParameters.OutputSamplePoints_Value[162] := 0.48000000000000043;
stInitData.ModelParameters.OutputSamplePoints_Value[163] := 0.48000000000000043;
stInitData.ModelParameters.OutputSamplePoints_Value[164] := 0.48000000000000043;
stInitData.ModelParameters.OutputSamplePoints_Value[165] := 0.59999999999999964;
stInitData.ModelParameters.OutputSamplePoints_Value[166] := 0.59999999999999964;
stInitData.ModelParameters.OutputSamplePoints_Value[167] := 0.59999999999999964;
stInitData.ModelParameters.OutputSamplePoints_Value[168] := 0.71999999999999975;
stInitData.ModelParameters.OutputSamplePoints_Value[169] := 0.71999999999999975;
stInitData.ModelParameters.OutputSamplePoints_Value[170] := 0.71999999999999975;
stInitData.ModelParameters.OutputSamplePoints_Value[171] := 0.83999999999999986;
stInitData.ModelParameters.OutputSamplePoints_Value[172] := 0.83999999999999986;
stInitData.ModelParameters.OutputSamplePoints_Value[173] := 0.83999999999999986;
stInitData.ModelParameters.OutputSamplePoints_Value[174] := 0.95999999999999996;
stInitData.ModelParameters.OutputSamplePoints_Value[175] := 0.95999999999999996;
stInitData.ModelParameters.OutputSamplePoints_Value[176] := 0.95999999999999996;
stInitData.ModelParameters.OutputSamplePoints_Value[177] := 1.0800000000000001;
stInitData.ModelParameters.OutputSamplePoints_Value[178] := 1.0800000000000001;
stInitData.ModelParameters.OutputSamplePoints_Value[179] := 1.0800000000000001;
stInitData.ModelParameters.OutputSamplePoints_Value[180] := 1.2000000000000002;
stInitData.ModelParameters.OutputSamplePoints_Value[181] := 1.2000000000000002;
stInitData.ModelParameters.OutputSamplePoints_Value[182] := 1.2000000000000002;
stInitData.ModelParameters.OutputSamplePoints_Value[183] := 1.3200000000000003;
stInitData.ModelParameters.OutputSamplePoints_Value[184] := 1.3200000000000003;
stInitData.ModelParameters.OutputSamplePoints_Value[185] := 1.3200000000000003;
stInitData.ModelParameters.OutputSamplePoints_Value[186] := 1.4400000000000004;
stInitData.ModelParameters.OutputSamplePoints_Value[187] := 1.4400000000000004;
stInitData.ModelParameters.OutputSamplePoints_Value[188] := 1.4400000000000004;
stInitData.ModelParameters.OutputSamplePoints_Value[189] := 1.5599999999999996;
stInitData.ModelParameters.OutputSamplePoints_Value[190] := 1.5599999999999996;
stInitData.ModelParameters.OutputSamplePoints_Value[191] := 1.5599999999999996;
stInitData.ModelParameters.OutputSamplePoints_Value[192] := 1.6799999999999997;
stInitData.ModelParameters.OutputSamplePoints_Value[193] := 1.6799999999999997;
stInitData.ModelParameters.OutputSamplePoints_Value[194] := 1.6799999999999997;
stInitData.ModelParameters.OutputSamplePoints_Value[195] := 1.7999999999999998;
stInitData.ModelParameters.OutputSamplePoints_Value[196] := 1.7999999999999998;
stInitData.ModelParameters.OutputSamplePoints_Value[197] := 1.7999999999999998;
stInitData.ModelParameters.OutputSamplePoints_Value[198] := 1.9199999999999999;
stInitData.ModelParameters.OutputSamplePoints_Value[199] := 1.9199999999999999;
stInitData.ModelParameters.OutputSamplePoints_Value[200] := 1.9199999999999999;
stInitData.ModelParameters.OutputSamplePoints_Value[201] := 2.0399999999999991;
stInitData.ModelParameters.OutputSamplePoints_Value[202] := 2.0399999999999991;
stInitData.ModelParameters.OutputSamplePoints_Value[203] := 2.0399999999999991;
stInitData.ModelParameters.OutputSamplePoints_Value[204] := 2.1600000000000001;
stInitData.ModelParameters.OutputSamplePoints_Value[205] := 2.1600000000000001;
stInitData.ModelParameters.OutputSamplePoints_Value[206] := 2.1600000000000001;
stInitData.ModelParameters.OutputSamplePoints_Value[207] := 2.2799999999999994;
stInitData.ModelParameters.OutputSamplePoints_Value[208] := 2.2799999999999994;
stInitData.ModelParameters.OutputSamplePoints_Value[209] := 2.2799999999999994;
stInitData.ModelParameters.OutputSamplePoints_Value[210] := 2.4000000000000004;
stInitData.ModelParameters.OutputSamplePoints_Value[211] := 2.4000000000000004;
stInitData.ModelParameters.OutputSamplePoints_Value[212] := 2.4000000000000004;
stInitData.ModelParameters.OutputSamplePoints_Value[213] := 2.5199999999999996;
stInitData.ModelParameters.OutputSamplePoints_Value[214] := 2.5199999999999996;
stInitData.ModelParameters.OutputSamplePoints_Value[215] := 2.5199999999999996;
stInitData.ModelParameters.OutputSamplePoints_Value[216] := 2.6400000000000006;
stInitData.ModelParameters.OutputSamplePoints_Value[217] := 2.6400000000000006;
stInitData.ModelParameters.OutputSamplePoints_Value[218] := 2.6400000000000006;
stInitData.ModelParameters.OutputSamplePoints_Value[219] := 2.7599999999999998;
stInitData.ModelParameters.OutputSamplePoints_Value[220] := 2.7599999999999998;
stInitData.ModelParameters.OutputSamplePoints_Value[221] := 2.7599999999999998;
stInitData.ModelParameters.OutputSamplePoints_Value[222] := 2.8800000000000008;
stInitData.ModelParameters.OutputSamplePoints_Value[223] := 2.8800000000000008;
stInitData.ModelParameters.OutputSamplePoints_Value[224] := 2.8800000000000008;
stInitData.ModelParameters.OutputSamplePoints_Value[225] := 3;
stInitData.ModelParameters.OutputSamplePoints_Value[226] := 3;
stInitData.ModelParameters.OutputSamplePoints_Value[227] := 3;
stInitData.ModelParameters.OutputSamplePoints_Value[228] := 3.1199999999999992;
stInitData.ModelParameters.OutputSamplePoints_Value[229] := 3.1199999999999992;
stInitData.ModelParameters.OutputSamplePoints_Value[230] := 3.1199999999999992;
stInitData.ModelParameters.OutputSamplePoints_Value[231] := 3.2400000000000002;
stInitData.ModelParameters.OutputSamplePoints_Value[232] := 3.2400000000000002;
stInitData.ModelParameters.OutputSamplePoints_Value[233] := 3.2400000000000002;
stInitData.ModelParameters.OutputSamplePoints_Value[234] := 3.3599999999999994;
stInitData.ModelParameters.OutputSamplePoints_Value[235] := 3.3599999999999994;
stInitData.ModelParameters.OutputSamplePoints_Value[236] := 3.3599999999999994;
stInitData.ModelParameters.OutputSamplePoints_Value[237] := 3.4800000000000004;
stInitData.ModelParameters.OutputSamplePoints_Value[238] := 3.4800000000000004;
stInitData.ModelParameters.OutputSamplePoints_Value[239] := 3.4800000000000004;
stInitData.ModelParameters.OutputSamplePoints_Value[240] := 3.5999999999999996;
stInitData.ModelParameters.OutputSamplePoints_Value[241] := 3.5999999999999996;
stInitData.ModelParameters.OutputSamplePoints_Value[242] := 3.5999999999999996;
stInitData.ModelParameters.OutputSamplePoints_Value[243] := 3.7200000000000006;
stInitData.ModelParameters.OutputSamplePoints_Value[244] := 3.7200000000000006;
stInitData.ModelParameters.OutputSamplePoints_Value[245] := 3.7200000000000006;
stInitData.ModelParameters.OutputSamplePoints_Value[246] := 3.8399999999999999;
stInitData.ModelParameters.OutputSamplePoints_Value[247] := 3.8399999999999999;
stInitData.ModelParameters.OutputSamplePoints_Value[248] := 3.8399999999999999;
stInitData.ModelParameters.OutputSamplePoints_Value[249] := 3.9600000000000009;
stInitData.ModelParameters.OutputSamplePoints_Value[250] := 3.9600000000000009;
stInitData.ModelParameters.OutputSamplePoints_Value[251] := 3.9600000000000009;
stInitData.ModelParameters.OutputSamplePoints_Value[252] := 4.0800000000000001;
stInitData.ModelParameters.OutputSamplePoints_Value[253] := 4.0800000000000001;
stInitData.ModelParameters.OutputSamplePoints_Value[254] := 4.0800000000000001;
stInitData.ModelParameters.OutputSamplePoints_Value[255] := 4.1999999999999993;
stInitData.ModelParameters.OutputSamplePoints_Value[256] := 4.1999999999999993;
stInitData.ModelParameters.OutputSamplePoints_Value[257] := 4.1999999999999993;
stInitData.ModelParameters.OutputSamplePoints_Value[258] := 4.3200000000000003;
stInitData.ModelParameters.OutputSamplePoints_Value[259] := 4.3200000000000003;
stInitData.ModelParameters.OutputSamplePoints_Value[260] := 4.3200000000000003;
stInitData.ModelParameters.OutputSamplePoints_Value[261] := 4.4399999999999995;
stInitData.ModelParameters.OutputSamplePoints_Value[262] := 4.4399999999999995;
stInitData.ModelParameters.OutputSamplePoints_Value[263] := 4.4399999999999995;
stInitData.ModelParameters.OutputSamplePoints_Value[264] := 4.5600000000000005;
stInitData.ModelParameters.OutputSamplePoints_Value[265] := 4.5600000000000005;
stInitData.ModelParameters.OutputSamplePoints_Value[266] := 4.5600000000000005;
stInitData.ModelParameters.OutputSamplePoints_Value[267] := 4.6799999999999997;
stInitData.ModelParameters.OutputSamplePoints_Value[268] := 4.6799999999999997;
stInitData.ModelParameters.OutputSamplePoints_Value[269] := 4.6799999999999997;
stInitData.ModelParameters.OutputSamplePoints_Value[270] := 4.8000000000000007;
stInitData.ModelParameters.OutputSamplePoints_Value[271] := 4.8000000000000007;
stInitData.ModelParameters.OutputSamplePoints_Value[272] := 4.8000000000000007;
stInitData.ModelParameters.OutputSamplePoints_Value[273] := 4.9199999999999999;
stInitData.ModelParameters.OutputSamplePoints_Value[274] := 4.9199999999999999;
stInitData.ModelParameters.OutputSamplePoints_Value[275] := 4.9199999999999999;
stInitData.ModelParameters.OutputSamplePoints_Value[276] := 5.0399999999999991;
stInitData.ModelParameters.OutputSamplePoints_Value[277] := 5.0399999999999991;
stInitData.ModelParameters.OutputSamplePoints_Value[278] := 5.0399999999999991;
stInitData.ModelParameters.OutputSamplePoints_Value[279] := 5.1600000000000001;
stInitData.ModelParameters.OutputSamplePoints_Value[280] := 5.1600000000000001;
stInitData.ModelParameters.OutputSamplePoints_Value[281] := 5.1600000000000001;
stInitData.ModelParameters.OutputSamplePoints_Value[282] := 5.2799999999999994;
stInitData.ModelParameters.OutputSamplePoints_Value[283] := 5.2799999999999994;
stInitData.ModelParameters.OutputSamplePoints_Value[284] := 5.2799999999999994;
stInitData.ModelParameters.OutputSamplePoints_Value[285] := 5.4000000000000004;
stInitData.ModelParameters.OutputSamplePoints_Value[286] := 5.4000000000000004;
stInitData.ModelParameters.OutputSamplePoints_Value[287] := 5.4000000000000004;
stInitData.ModelParameters.OutputSamplePoints_Value[288] := 5.5199999999999996;
stInitData.ModelParameters.OutputSamplePoints_Value[289] := 5.5199999999999996;
stInitData.ModelParameters.OutputSamplePoints_Value[290] := 5.5199999999999996;
stInitData.ModelParameters.OutputSamplePoints_Value[291] := 5.6400000000000006;
stInitData.ModelParameters.OutputSamplePoints_Value[292] := 5.6400000000000006;
stInitData.ModelParameters.OutputSamplePoints_Value[293] := 5.6400000000000006;
stInitData.ModelParameters.OutputSamplePoints_Value[294] := 5.7599999999999998;
stInitData.ModelParameters.OutputSamplePoints_Value[295] := 5.7599999999999998;
stInitData.ModelParameters.OutputSamplePoints_Value[296] := 5.7599999999999998;
stInitData.ModelParameters.OutputSamplePoints_Value[297] := 5.8800000000000008;
stInitData.ModelParameters.OutputSamplePoints_Value[298] := 5.8800000000000008;
stInitData.ModelParameters.OutputSamplePoints_Value[299] := 5.8800000000000008;
stInitData.ModelParameters.OutputSamplePoints_Value[300] := 6;
stInitData.ModelParameters.OutputSamplePoints_Value[301] := 6;
stInitData.ModelParameters.OutputSamplePoints_Value[302] := 6;
stInitData.ModelParameters.H_IC := 1;
stInitData.ModelParameters.H_UpperSat := 1.7976931348623157e+308;
stInitData.ModelParameters.H_LowerSat := 0;
stInitData.ModelParameters.Ke_Gain := 0.01;
stInitData.ModelParameters.Kec_Gain := 0.01;
stInitData.ModelParameters.K1_Gain := 0.5;
stInitData.ModelParameters.K2_Gain := 0.01;
stInitData.ModelParameters.kp0_Value := 0.208480938103529;
stInitData.ModelParameters.ki0_Value := 0.031284128435613602;
stInitData.ModelParameters.Integrator1_IC := 0;
stInitData.ContextInfoArr_0_TaskOidHdr.indexGroup := 0;
stInitData.ContextInfoArr_0_TaskOidHdr.indexOffset := 16#03002060;
stInitData.ContextInfoArr_0_TaskOidHdr.cbData := SIZEOF(stInitData.ContextInfoArr_0_TaskOid);
stInitData.ContextInfoArr_0_TaskPriorityHdr.indexGroup := 0;
stInitData.ContextInfoArr_0_TaskPriorityHdr.indexOffset := 16#03002070;
stInitData.ContextInfoArr_0_TaskPriorityHdr.cbData := SIZEOF(stInitData.ContextInfoArr_0_TaskPriority);
stInitData.ContextInfoArr_0_TaskCycleTimeNsHdr.indexGroup := 0;
stInitData.ContextInfoArr_0_TaskCycleTimeNsHdr.indexOffset := 16#03002080;
stInitData.ContextInfoArr_0_TaskCycleTimeNsHdr.cbData := SIZEOF(stInitData.ContextInfoArr_0_TaskCycleTimeNs);
stInitData.ContextInfoArr_0_TaskPortHdr.indexGroup := 0;
stInitData.ContextInfoArr_0_TaskPortHdr.indexOffset := 16#03002090;
stInitData.ContextInfoArr_0_TaskPortHdr.cbData := SIZEOF(stInitData.ContextInfoArr_0_TaskPort);
stInitData.ContextInfoArr_0_TaskSortOrderHdr.indexGroup := 0;
stInitData.ContextInfoArr_0_TaskSortOrderHdr.indexOffset := 16#030020b0;
stInitData.ContextInfoArr_0_TaskSortOrderHdr.cbData := SIZEOF(stInitData.ContextInfoArr_0_TaskSortOrder);
stInitData.Header.cbData := SIZEOF(stInitData)-SIZEOF(stInitData.Header);
stInitData.Header.uiElmCnt := 10;


// set pointer to InitData structure
SetInitDataInfo(ADR(stInitData));

// set DataArea information
SetDataAreaInfo(ADR(arrDataAreas),2);
arrDataAreas[1].nDataAreaId := 0;
arrDataAreas[1].nSize := SIZEOF(stInput);
arrDataAreas[1].pPlcVar := ADR(stInput);
arrDataAreas[1].pModuleProcImg := 0;
arrDataAreas[1].eDataAreaType := E_TcMatSimDataAreaType.InputDst;
arrDataAreas[2].nDataAreaId := 1;
arrDataAreas[2].nSize := SIZEOF(stOutput);
arrDataAreas[2].pPlcVar := ADR(stOutput);
arrDataAreas[2].pModuleProcImg := 0;
arrDataAreas[2].eDataAreaType := E_TcMatSimDataAreaType.OutputSrc;


// initialize basic interface pointers and return
FB_init := SUCCEEDED(Init(oid));
                  
                
END_METHOD

METHOD Execute : HRESULT
                  
IF (SUCCEEDED(hResult)) THEN
  hResult := VerifyParameters();
END_IF

// update DataArea information
SetDataAreaInfo(ADR(arrDataAreas),2);
arrDataAreas[1].nDataAreaId := 0;
arrDataAreas[1].nSize := SIZEOF(stInput);
arrDataAreas[1].pPlcVar := ADR(stInput);
arrDataAreas[1].pModuleProcImg := 0;
arrDataAreas[1].eDataAreaType := E_TcMatSimDataAreaType.InputDst;
arrDataAreas[2].nDataAreaId := 1;
arrDataAreas[2].nSize := SIZEOF(stOutput);
arrDataAreas[2].pPlcVar := ADR(stOutput);
arrDataAreas[2].pModuleProcImg := 0;
arrDataAreas[2].eDataAreaType := E_TcMatSimDataAreaType.OutputSrc;

	
// call base method
Execute := SUPER^.Execute();
                  
                
END_METHOD

{attribute 'object_name' := 'VerifyParameters'}
METHOD VerifyParameters : HRESULT
  VAR
    moduleCallByParam : TctModuleCallByType;
  END_VAR
                  
IF (bParametersVerified) THEN
  VerifyParameters := Tc2_System.E_HRESULTAdsErr.HRESULT_ADS_NOERROR;
ELSE
  VerifyParameters := GetObjPara(stInitData.CallByHdr.indexOffset,SIZEOF(moduleCallByParam),ADR(moduleCallByParam));
  
  // check the "CallBy" parameter to be set to "Module"
  IF (SUCCEEDED(VerifyParameters) AND (moduleCallByParam <> TctModuleCallByType.Module)) THEN
      VerifyParameters := Tc2_System.E_HRESULTAdsErr.INVALIDPARM;
  END_IF
  
  // set the parameters verified flag
  bParametersVerified := SUCCEEDED(VerifyParameters);
END_IF
                  
                
END_METHOD

PROPERTY InitData : ST_AdaptiveModelInitData
GET
                    InitData := stInitData;
                  
END_GET
SET
                    stInitData := InitData;
                  
END_SET
END_PROPERTY

PROPERTY CallBy_Startup : TctModuleCallByType
GET
						CallBy_Startup := stInitData.CallBy;
					
END_GET
SET
						stInitData.CallBy := CallBy_Startup;
					
END_SET
END_PROPERTY

PROPERTY ExecutionSequence_Startup : TctModuleExecutionSequenceType
GET
						ExecutionSequence_Startup := stInitData.ExecutionSequence;
					
END_GET
SET
						stInitData.ExecutionSequence := ExecutionSequence_Startup;
					
END_SET
END_PROPERTY

PROPERTY StepSize_Startup : TctStepSizeType
GET
						StepSize_Startup := stInitData.StepSize;
					
END_GET
SET
						stInitData.StepSize := StepSize_Startup;
					
END_SET
END_PROPERTY

PROPERTY ExecuteModelCode_Startup : BOOL
GET
						ExecuteModelCode_Startup := stInitData.ExecuteModelCode;
					
END_GET
SET
						stInitData.ExecuteModelCode := ExecuteModelCode_Startup;
					
END_SET
END_PROPERTY

PROPERTY ModelParameters_Startup : P_AdaptiveModel_T
GET
						ModelParameters_Startup := stInitData.ModelParameters;
					
END_GET
SET
						stInitData.ModelParameters := ModelParameters_Startup;
					
END_SET
END_PROPERTY

PROPERTY ContextInfoArr_0_TaskOid_Startup : OTCID
GET
						ContextInfoArr_0_TaskOid_Startup := stInitData.ContextInfoArr_0_TaskOid;
					
END_GET
SET
						stInitData.ContextInfoArr_0_TaskOid := ContextInfoArr_0_TaskOid_Startup;
					
END_SET
END_PROPERTY

PROPERTY ContextInfoArr_0_TaskPriority_Startup : UDINT
GET
						ContextInfoArr_0_TaskPriority_Startup := stInitData.ContextInfoArr_0_TaskPriority;
					
END_GET
SET
						stInitData.ContextInfoArr_0_TaskPriority := ContextInfoArr_0_TaskPriority_Startup;
					
END_SET
END_PROPERTY

PROPERTY ContextInfoArr_0_TaskCycleTimeNs_Startup : UDINT
GET
						ContextInfoArr_0_TaskCycleTimeNs_Startup := stInitData.ContextInfoArr_0_TaskCycleTimeNs;
					
END_GET
SET
						stInitData.ContextInfoArr_0_TaskCycleTimeNs := ContextInfoArr_0_TaskCycleTimeNs_Startup;
					
END_SET
END_PROPERTY

PROPERTY ContextInfoArr_0_TaskPort_Startup : UINT
GET
						ContextInfoArr_0_TaskPort_Startup := stInitData.ContextInfoArr_0_TaskPort;
					
END_GET
SET
						stInitData.ContextInfoArr_0_TaskPort := ContextInfoArr_0_TaskPort_Startup;
					
END_SET
END_PROPERTY

PROPERTY ContextInfoArr_0_TaskSortOrder_Startup : UDINT
GET
						ContextInfoArr_0_TaskSortOrder_Startup := stInitData.ContextInfoArr_0_TaskSortOrder;
					
END_GET
SET
						stInitData.ContextInfoArr_0_TaskSortOrder := ContextInfoArr_0_TaskSortOrder_Startup;
					
END_SET
END_PROPERTY

PROPERTY CallBy_Online : TctModuleCallByType
GET
						hResult := GetObjPara(16#00000000,sizeof(CallBy_Online),adr(CallBy_Online));
					
END_GET
SET
						hResult := SetObjPara(16#00000000,sizeof(CallBy_Online),adr(CallBy_Online));
					
END_SET
END_PROPERTY

PROPERTY ExecutionSequence_Online : TctModuleExecutionSequenceType
GET
						hResult := GetObjPara(16#00000001,sizeof(ExecutionSequence_Online),adr(ExecutionSequence_Online));
					
END_GET
SET
						hResult := SetObjPara(16#00000001,sizeof(ExecutionSequence_Online),adr(ExecutionSequence_Online));
					
END_SET
END_PROPERTY

PROPERTY StepSize_Online : TctStepSizeType
GET
						hResult := GetObjPara(16#00000002,sizeof(StepSize_Online),adr(StepSize_Online));
					
END_GET
SET
						hResult := SetObjPara(16#00000002,sizeof(StepSize_Online),adr(StepSize_Online));
					
END_SET
END_PROPERTY

PROPERTY MdlInitialized_Online : BOOL
GET
						hResult := GetObjPara(16#00000003,sizeof(MdlInitialized_Online),adr(MdlInitialized_Online));
					
END_GET
SET
						hResult := SetObjPara(16#00000003,sizeof(MdlInitialized_Online),adr(MdlInitialized_Online));
					
END_SET
END_PROPERTY

PROPERTY CycleUpdateExecuted_Online : BOOL
GET
						hResult := GetObjPara(16#00000004,sizeof(CycleUpdateExecuted_Online),adr(CycleUpdateExecuted_Online));
					
END_GET
SET
						hResult := SetObjPara(16#00000004,sizeof(CycleUpdateExecuted_Online),adr(CycleUpdateExecuted_Online));
					
END_SET
END_PROPERTY

PROPERTY ModuleInfo_Online : TctModuleInfoType
GET
						hResult := GetObjPara(16#00000005,sizeof(ModuleInfo_Online),adr(ModuleInfo_Online));
					
END_GET
SET
						hResult := SetObjPara(16#00000005,sizeof(ModuleInfo_Online),adr(ModuleInfo_Online));
					
END_SET
END_PROPERTY

PROPERTY ModuleBuildInfo_Online : TctModuleBuildInfoType
GET
						hResult := GetObjPara(16#00000006,sizeof(ModuleBuildInfo_Online),adr(ModuleBuildInfo_Online));
					
END_GET
SET
						hResult := SetObjPara(16#00000006,sizeof(ModuleBuildInfo_Online),adr(ModuleBuildInfo_Online));
					
END_SET
END_PROPERTY

PROPERTY ExecuteModelCode_Online : BOOL
GET
						hResult := GetObjPara(16#00000007,sizeof(ExecuteModelCode_Online),adr(ExecuteModelCode_Online));
					
END_GET
SET
						hResult := SetObjPara(16#00000007,sizeof(ExecuteModelCode_Online),adr(ExecuteModelCode_Online));
					
END_SET
END_PROPERTY

PROPERTY SimulinkTime_Online : LREAL
GET
						hResult := GetObjPara(16#00000008,sizeof(SimulinkTime_Online),adr(SimulinkTime_Online));
					
END_GET
SET
						hResult := SetObjPara(16#00000008,sizeof(SimulinkTime_Online),adr(SimulinkTime_Online));
					
END_SET
END_PROPERTY

PROPERTY Input_Online : ExtU_AdaptiveModel_T
GET
						hResult := GetObjPara(16#80000000,sizeof(Input_Online),adr(Input_Online));
					
END_GET
SET
						hResult := SetObjPara(16#80000000,sizeof(Input_Online),adr(Input_Online));
					
END_SET
END_PROPERTY

PROPERTY ModelParameters_Online : P_AdaptiveModel_T
GET
						hResult := GetObjPara(16#83000000,sizeof(ModelParameters_Online),adr(ModelParameters_Online));
					
END_GET
SET
						hResult := SetObjPara(16#83000000,sizeof(ModelParameters_Online),adr(ModelParameters_Online));
					
END_SET
END_PROPERTY

PROPERTY ContextInfoArr_0_TaskOid_Online : OTCID
GET
						hResult := GetObjPara(16#03002060,sizeof(ContextInfoArr_0_TaskOid_Online),adr(ContextInfoArr_0_TaskOid_Online));
					
END_GET
SET
						hResult := SetObjPara(16#03002060,sizeof(ContextInfoArr_0_TaskOid_Online),adr(ContextInfoArr_0_TaskOid_Online));
					
END_SET
END_PROPERTY

PROPERTY ContextInfoArr_0_TaskPriority_Online : UDINT
GET
						hResult := GetObjPara(16#03002070,sizeof(ContextInfoArr_0_TaskPriority_Online),adr(ContextInfoArr_0_TaskPriority_Online));
					
END_GET
SET
						hResult := SetObjPara(16#03002070,sizeof(ContextInfoArr_0_TaskPriority_Online),adr(ContextInfoArr_0_TaskPriority_Online));
					
END_SET
END_PROPERTY

PROPERTY ContextInfoArr_0_TaskCycleTimeNs_Online : UDINT
GET
						hResult := GetObjPara(16#03002080,sizeof(ContextInfoArr_0_TaskCycleTimeNs_Online),adr(ContextInfoArr_0_TaskCycleTimeNs_Online));
					
END_GET
SET
						hResult := SetObjPara(16#03002080,sizeof(ContextInfoArr_0_TaskCycleTimeNs_Online),adr(ContextInfoArr_0_TaskCycleTimeNs_Online));
					
END_SET
END_PROPERTY

PROPERTY ContextInfoArr_0_TaskPort_Online : UINT
GET
						hResult := GetObjPara(16#03002090,sizeof(ContextInfoArr_0_TaskPort_Online),adr(ContextInfoArr_0_TaskPort_Online));
					
END_GET
SET
						hResult := SetObjPara(16#03002090,sizeof(ContextInfoArr_0_TaskPort_Online),adr(ContextInfoArr_0_TaskPort_Online));
					
END_SET
END_PROPERTY

PROPERTY ContextInfoArr_0_TaskSortOrder_Online : UDINT
GET
						hResult := GetObjPara(16#030020b0,sizeof(ContextInfoArr_0_TaskSortOrder_Online),adr(ContextInfoArr_0_TaskSortOrder_Online));
					
END_GET
SET
						hResult := SetObjPara(16#030020b0,sizeof(ContextInfoArr_0_TaskSortOrder_Online),adr(ContextInfoArr_0_TaskSortOrder_Online));
					
END_SET
END_PROPERTY
END_FUNCTION_BLOCK
